(* CODESYS project mobject-reports.library
   Company: mobject
   DefaultNamespace: mobject-reports
   Version: 0.3.0
   Placeholder: mobject-reports
   Author: mobject dev team
   Title: mobject-reports

Project tree, tasks and I/O mapping:
  libraries: mobject-core, 0.6.0 (mobject); Tc2_System, * (Beckhoff Automation GmbH); Tc2_Utilities, * (Beckhoff Automation GmbH); Tc3_Module, * (Beckhoff Automation GmbH)
  _Internal/
    Common/
      data type AppSystemInfoStructure
      data type TaskSystemInfoStructure
    Helper Functions/
      function GetAppSystemInfo [ST]
      function GetSymbolNameFromAny [ST]
      function GetTaskSystemInfo [ST]
    Interfaces/
      interface I_ReportGenerator: Generate
    PDFReport/
      Commands/
        function block ReportGenerateCommand [ST]: OnExecuting, OnInitializing, Setup
      DUT/
        data type PDFReportRequestStructure
        data type PDFReportResponseStructure
  PDFReport/
    function block PDFReport [ST]: Busy, CyclicCall, Done, Error, ErrorId, Generate
*)

// _Internal/Common/AppSystemInfoStructure
{attribute 'pack_mode' := '1'}
TYPE AppSystemInfoStructure :
STRUCT
	TaskCnt : UDINT;
	OnlineChangeCnt : UDINT;
	Flags : DWORD;
	AdsPort : UINT;
	BootDataLoaded : BOOL;
	OldBootData : BOOL;
	AppTimestamp : DT;
	KeepOutputsOnBP : BOOL;
	ShutdownInProgress : BOOL;
	LicensesPending : BOOL;
	BSODOccured : BOOL;
	LoggedIn : BOOL;
	AppName : STRING(63);
	ProjectName : STRING(63);
	PersistentStatus : EPlcPersistentStatus;
END_STRUCT
END_TYPE

// _Internal/Common/TaskSystemInfoStructure
{attribute 'pack_mode' := '1'}
TYPE TaskSystemInfoStructure :
STRUCT
	CycleTime : UDINT;
	Priority : UINT;
	AdsPort : UINT;
	CycleCount : UDINT;
	DcTaskTime : LINT;
	LastExecTime : UDINT;
	FirstCycle : BOOL; 
	CycleTimeExceeded : BOOL; 
	InCallAfterOutputUpdate : BOOL; 
	RTViolation : BOOL;
	TaskName : STRING(63);
END_STRUCT
END_TYPE

// _Internal/PDFReport/DUT/PDFReportRequestStructure
{attribute 'pack_mode' := '1'}
TYPE PDFReportRequestStructure :
STRUCT
	VariableName : T_MAXSTRING;
	LocalNetId : T_AmsNetId;
	LocalPort : UINT;
	TemplateName : T_MAXSTRING;
	FileName : T_MAXSTRING;
	FilePath : T_MAXSTRING;
	AppSystemInfo : AppSystemInfoStructure;
	TaskSystemInfo : TaskSystemInfoStructure;
END_STRUCT
END_TYPE

// _Internal/PDFReport/DUT/PDFReportResponseStructure
{attribute 'pack_mode' := '1'}
TYPE PDFReportResponseStructure :
STRUCT
	ResponseCode : UDINT;
END_STRUCT
END_TYPE

// _Internal/Helper Functions/GetAppSystemInfo
{attribute 'linkalways'} 
FUNCTION GetAppSystemInfo : AppSystemInfoStructure

GetAppSystemInfo.AdsPort := TwinCAT_SystemInfoVarList._AppInfo.AdsPort;
GetAppSystemInfo.AppName := TwinCAT_SystemInfoVarList._AppInfo.AppName;
GetAppSystemInfo.AppTimestamp :=TwinCAT_SystemInfoVarList. _AppInfo.AppTimestamp;
GetAppSystemInfo.BootDataLoaded := TwinCAT_SystemInfoVarList._AppInfo.BootDataLoaded;
GetAppSystemInfo.BSODOccured := TwinCAT_SystemInfoVarList._AppInfo.BSODOccured;
GetAppSystemInfo.Flags := TwinCAT_SystemInfoVarList._AppInfo.Flags;
GetAppSystemInfo.KeepOutputsOnBP := TwinCAT_SystemInfoVarList._AppInfo.KeepOutputsOnBP;
GetAppSystemInfo.LicensesPending := TwinCAT_SystemInfoVarList._AppInfo.LicensesPending;
GetAppSystemInfo.LoggedIn := TwinCAT_SystemInfoVarList._AppInfo.LoggedIn;
GetAppSystemInfo.OldBootData := TwinCAT_SystemInfoVarList._AppInfo.OldBootData;
GetAppSystemInfo.OnlineChangeCnt := TwinCAT_SystemInfoVarList._AppInfo.OnlineChangeCnt;
GetAppSystemInfo.PersistentStatus := TwinCAT_SystemInfoVarList._AppInfo.PersistentStatus;
GetAppSystemInfo.ProjectName := TwinCAT_SystemInfoVarList._AppInfo.ProjectName;
GetAppSystemInfo.ShutdownInProgress := TwinCAT_SystemInfoVarList._AppInfo.ShutdownInProgress;
GetAppSystemInfo.TaskCnt := TwinCAT_SystemInfoVarList._AppInfo.TaskCnt;

END_FUNCTION

// _Internal/Helper Functions/GetSymbolNameFromAny
{attribute 'linkalways'} 
FUNCTION GetSymbolNameFromAny : T_MAXSTRING
VAR_INPUT
	Symbol : ANY;
END_VAR
VAR
	hr : HRESULT;
	appInfo : ITcIecApplicationInfo;

	symbolNameLength : UDINT;	
	pSymbolName : POINTER TO BYTE;
	pSymbolNameAsString : POINTER TO STRING;
END_VAR

REPEAT
	
	// if it's not an enum then exit
	IF Symbol.TypeClass <> __SYSTEM.TYPE_CLASS.TYPE_USERDEF THEN 
		EXIT; 
	END_IF
	
	// ------------------------------------------------
	// Get the application info object
	// ------------------------------------------------	
	IF TwinCAT_SystemInfoVarList._AppInfo.ObjId = 0 THEN 
		EXIT; 
	END_IF

	// get the application info object
	hr := FW_ObjMgr_GetObjectInstance(TwinCAT_SystemInfoVarList._AppInfo.ObjId, TC_GLOBAL_IID_LIST.IID_ITcIecApplicationInfo, ADR(appInfo));
	IF FAILED(hr) THEN 
		EXIT; 
	END_IF
	
	// ------------------------------------------------
	// Get the symbol name based on the symbol address
	// ------------------------------------------------
	
	// get the symbol name length
	hr := appInfo.GetSymbolNameByAddress(0, Symbol.pValue, symbolNameLength, 0);
	IF symbolNameLength = 0 THEN 
		EXIT; 
	END_IF
	
	// make string to hold the symbol name
	pSymbolName := __NEW(BYTE,symbolNameLength);
	
	// get symbol name by address
	hr := appInfo.GetSymbolNameByAddress(symbolNameLength, Symbol.pValue, symbolNameLength, pSymbolName);
	IF FAILED(hr) THEN 
		EXIT; 
	END_IF
	
	// convert the pointer to a pointer to string;
	pSymbolNameAsString := pSymbolName;
	
UNTIL TRUE // this allows us to exit out of the repeat at any point.
END_REPEAT

IF pSymbolNameAsString <> 0 THEN
	GetSymbolNameFromAny := pSymbolNameAsString^;
END_IF

// tidy app info before leaving
FW_SafeRelease(ADR(appInfo));

// tidy symbol name before leaving
IF pSymbolName <> 0 THEN
	__DELETE(pSymbolName);
END_IF

END_FUNCTION

// _Internal/Helper Functions/GetTaskSystemInfo
{attribute 'linkalways'} 
FUNCTION GetTaskSystemInfo : TaskSystemInfoStructure
VAR
	getTaskIndex : GETCURTASKINDEX;
	taskInfo : PlcTaskSystemInfo;
END_VAR

getTaskIndex();
taskInfo := TwinCAT_SystemInfoVarList._TaskInfo[getTaskIndex.index];
GetTaskSystemInfo.AdsPort := taskInfo.AdsPort;
GetTaskSystemInfo.CycleCount := taskInfo.CycleCount;
GetTaskSystemInfo.CycleTime := taskInfo.CycleTime;
GetTaskSystemInfo.CycleTimeExceeded := taskInfo.CycleTimeExceeded;
GetTaskSystemInfo.DcTaskTime := taskInfo.DcTaskTime;
GetTaskSystemInfo.FirstCycle := taskInfo.FirstCycle;
GetTaskSystemInfo.InCallAfterOutputUpdate := taskInfo.InCallAfterOutputUpdate;
GetTaskSystemInfo.LastExecTime := taskInfo.LastExecTime;
GetTaskSystemInfo.Priority := taskInfo.Priority;
GetTaskSystemInfo.RTViolation := taskInfo.RTViolation;
GetTaskSystemInfo.TaskName := taskInfo.TaskName;

END_FUNCTION

// _Internal/Interfaces/I_ReportGenerator
INTERFACE I_ReportGenerator

METHOD PUBLIC Generate
VAR_INPUT
	SourceData : ANY;
	TemplateName : T_MAXSTRING;
	FileName : T_MAXSTRING;
	FilePath : T_MAXSTRING;
END_VAR
END_METHOD

END_INTERFACE

// _Internal/PDFReport/Commands/ReportGenerateCommand
{attribute 'linkalways'} 
{attribute 'no_explicit_call' := 'This FB is a CLASS and must be accessed using methods or properties'}
{attribute 'enable_dynamic_creation'}
FUNCTION_BLOCK ReportGenerateCommand EXTENDS AsyncCommand
VAR
	requestData : PDFReportRequestStructure;
	responseData : PDFReportResponseStructure;
	getLocalAmsNetId : FB_GetLocalAmsNetId;
	adsReadWriter : ADSRDWRTEX;
	state : (GET_LOCAL_DETAILS, SEND_REQUEST) := GET_LOCAL_DETAILS;
END_VAR
VAR CONSTANT
	MOBJECT_REPORT_APP_AMSPORT : T_AmsPort := 27272;
	MOBJECT_REPORT_APP_GROUP : UDINT := 10;
	MOBJECT_REPORT_APP_OFFSET : UDINT := 100;
	MOBJECT_REPORT_APP_OK : UDINT := 200;
END_VAR

METHOD PROTECTED OnExecuting
VAR_INPUT
	StateControl : I_AsyncCommandStateControl;
END_VAR
CASE state OF
	
	GET_LOCAL_DETAILS : 
	
		getLocalAmsNetId(bExecute := TRUE);
		IF getLocalAmsNetId.bBusy THEN
			RETURN;
		END_IF
		
		IF getLocalAmsNetId.bError THEN
			StateControl.Error(getLocalAmsNetId.nErrId);
			RETURN;
		END_IF
		
		requestData.LocalNetId := getLocalAmsNetId.AddrString;
		requestData.LocalPort := TwinCAT_SystemInfoVarList._AppInfo.AdsPort;;
		
		state := SEND_REQUEST;
		
	SEND_REQUEST:
			
		AdsReadWriter(
			NETID := , 
			PORT := MOBJECT_REPORT_APP_AMSPORT, 
			IDXGRP := MOBJECT_REPORT_APP_GROUP,
			IDXOFFS := MOBJECT_REPORT_APP_OFFSET,
			WRITELEN := SIZEOF(requestData), 
			READLEN := SIZEOF(responseData), 
			SRCADDR := ADR(requestData),  
			DESTADDR := ADR(responseData), 
			WRTRD := TRUE
		);
		
		IF AdsReadWriter.BUSY THEN
			RETURN;
		END_IF
		
		IF AdsReadWriter.ERR THEN
			StateControl.Error(AdsReadWriter.ERRID);
			RETURN;
		END_IF
		
//		IF responseData.ResponseCode <> MOBJECT_REPORT_APP_OK THEN
//			StateControl.Error(responseData.ResponseCode);
//			RETURN;
//		END_IF
		
		StateControl.Next();
	
END_CASE
END_METHOD

METHOD PROTECTED OnInitializing
VAR_INPUT
	StateControl : I_AsyncCommandStateControl;
END_VAR
getLocalAmsNetId(bExecute := FALSE);
AdsReadWriter(WRTRD	:= FALSE);
StateControl.Next();
END_METHOD

METHOD PUBLIC Setup
VAR_INPUT
	SourceData : ANY;
	TemplateName : T_MAXSTRING;
	FileName : T_MAXSTRING;
	FilePath : T_MAXSTRING;
END_VAR
IF NOT Busy THEN
	requestData.VariableName := GetSymbolNameFromAny(SourceData); 
	requestData.TemplateName := TemplateName;
	requestData.FileName := FileName;
	requestData.FilePath := FilePath;
	requestData.AppSystemInfo := GetAppSystemInfo();
	requestData.TaskSystemInfo := GetTaskSystemInfo();
END_IF
END_METHOD

END_FUNCTION_BLOCK

// PDFReport/PDFReport
{attribute 'linkalways'} 
{attribute 'no_explicit_call' := 'This FB is a CLASS and must be accessed using methods or properties'}
{attribute 'enable_dynamic_creation'}
FUNCTION_BLOCK PDFReport IMPLEMENTS I_ReportGenerator
VAR
	reportGenerateCommand : ReportGenerateCommand;
END_VAR

PROPERTY PUBLIC Busy : BOOL
GET
Busy := reportGenerateCommand.Busy;
END_GET
END_PROPERTY

METHOD PUBLIC CyclicCall
VAR_INPUT
END_VAR
IF reportGenerateCommand.Busy THEN
	reportGenerateCommand.CyclicCall();
END_IF
END_METHOD

PROPERTY PUBLIC Done : BOOL
GET
Done := reportGenerateCommand.Done;
END_GET
END_PROPERTY

PROPERTY PUBLIC Error : BOOL
GET
Error := reportGenerateCommand.Error;
END_GET
END_PROPERTY

PROPERTY PUBLIC ErrorId : UDINT
GET
ErrorId := reportGenerateCommand.ErrorId;
END_GET
END_PROPERTY

METHOD PUBLIC Generate
VAR_INPUT
	SourceData : ANY; // SourceData must be a Structure DUT
	TemplateName : T_MAXSTRING;
	FileName : T_MAXSTRING;
	FilePath : T_MAXSTRING;
END_VAR
reportGenerateCommand.Setup(
	SourceData := SourceData,
	TemplateName := TemplateName,
	FileName := FileName,
	FilePath := FilePath
);

reportGenerateCommand.Execute();
END_METHOD

END_FUNCTION_BLOCK
